// TwinCAT 3 PLC project Untitled1
// ProgramVersion: 3.1.4023.0
// libraries:
//   Tc2_MC2, * (Beckhoff Automation GmbH)
//   Tc2_Standard, * (Beckhoff Automation GmbH)
//   Tc2_System, * (Beckhoff Automation GmbH)
//   Tc3_Module, * (Beckhoff Automation GmbH)
// project tree:
//   DUTs/ st_axisInput.TcDUT, st_axisInterface.TcDUT, st_axisOutput.TcDUT
//   / GlobalTextList.TcGTLO, PlcTask.TcTTO, Visualization Manager.TcVMO (not stored)
//   GVLs/ GVL_Axis.TcGVL
//   POUs/ Fb_Motion.TcPOU, MAIN.TcPOU
//   VISUs/ VISU_1.TcVIS, VISU_2.TcVIS
// real-time tasks:
//   TASK PlcTask: cycle T#10ms, priority 20, ADS port 350
// motion (NC):
//   TASK NC-Task 1 SAF: cycle T#2ms, priority 4, ADS port 501
//   TASK NC-Task 1 SVB: cycle T#10ms, priority 8, ADS port 511
//   AXIS Axis 1 (id 1)
//     OtherSettings: AllowMotionCmdToSlave=true
//     encoder EncType=1
//     drive DrvType=5
//       Analog: TorqueSetpointScale=10, ScaleFactorActTorque=0.1
//     controller CtrType=1
//       CtrPara: PriorControlFactor=1
//         Observer: BandWidth=20
// variable links:
//   Untitled1/Untitled1 Instance <-> NC-Task 1 SAF/Axes/Axis 1
//     PlcTask Inputs/GVL_Axis.Axis1.NcToPlc <-> Outputs/ToPlc
//     PlcTask Outputs/GVL_Axis.Axis1.PlcToNc <-> Inputs/FromPlc

CONFIGURATION Untitled1
    RESOURCE PLC ON TwinCAT3
        TASK PlcTask(INTERVAL := T#10ms, PRIORITY := 20);
        PROGRAM MAIN WITH PlcTask : MAIN;
    END_RESOURCE
END_CONFIGURATION

// ---- DUTs/st_axisInput.TcDUT
TYPE st_axisInput :
STRUCT
	

	bPowerEnable	:	BOOL;
	bMoveAbs		:	BOOL;
	bStop			:	BOOL;
	bReset			:	BOOL;
	
	
	fOverride	:	LREAL;
	fPosition	:	LREAL;
	fVelocity	:	LREAL;

	
	
	

END_STRUCT
END_TYPE

// ---- DUTs/st_axisInterface.TcDUT
TYPE st_axisInterface :
STRUCT
	

IN	:	st_axisInput;
OUT	:	st_axisOutput;


END_STRUCT
END_TYPE

// ---- DUTs/st_axisOutput.TcDUT
TYPE st_axisOutput :
STRUCT
	

	bPowerEnabled	:	BOOL;
	bPowerErr		:	BOOL;

	bMoveAbsDone	:	BOOL;
	bMoveAbsBusy	:	BOOL;
	bMoveAbsErr		:	BOOL;
	
	
	bStopDone		:	BOOL;
	bStopActive		:	BOOL;
	bStopErr		:	BOOL;
	
	bResetDone		:	BOOL;
	bResetErr		:	BOOL;

END_STRUCT
END_TYPE

// ---- GVLs/GVL_Axis.TcGVL
{attribute 'qualified_only'}
VAR_GLOBAL
	

	Axis1	:	AXIS_REF;		//	1. Motor
	
	stAxis1	:	st_axisInterface;
	
	
	Axis2	:	AXIS_REF;		//	2.Motor

	stAxis2	:	st_axisInterface;

END_VAR

// ---- POUs/MAIN.TcPOU
PROGRAM MAIN
VAR
	FbMotion1: Fb_Motion;
	FbMotion2: Fb_Motion;
	nState: INT;
	bButon: BOOL;
	T1: TON;
	T2: TON;
	T3: TON;
	bResetButon	:	BOOL;
	rtrig1: R_TRIG;
	bCounter: BOOL;
	nCounter: INT;
	sMsgInfo: STRING;
	sMsgVelo: STRING;
	sMsgPosition: STRING;
	fPositionVisu: LREAL;
END_VAR



ACT_Motion();
ACT_Visu();







FbMotion1(Axis:=GVL_Axis.Axis1 , stAxis:=GVL_Axis.stAxis1 );
//FbMotion2(Axis:=GVL_Axis.Axis2 , stAxis:=GVL_Axis.stAxis2 );

ACTION ACT_Motion:


rtrig1(CLK:=bCounter , Q=> );


CASE nState OF
	



	0:
	
		IF bButon THEN
			
		GVL_Axis.stAxis1.IN.bPowerEnable	:=	TRUE;
		GVL_Axis.stAxis1.IN.fOverride	:=	100.0;
		GVL_Axis.stAxis1.IN.bStop	:=	FALSE;	
		GVL_Axis.stAxis1.IN.bMoveAbs	:=	FALSE;
		nState := 1;
		
		END_IF
	
		
	1:
		IF	bButon	
		AND NOT GVL_Axis.stAxis1.OUT.bPowerErr
		AND NOT GVL_Axis.stAxis1.OUT.bStopActive 
		AND GVL_Axis.stAxis1.OUT.bPowerEnabled THEN
		
			nState := 10;
			
		END_IF
	
	
	10:
		
		GVL_Axis.stAxis1.IN.fPosition	:=	5000;
		GVL_Axis.stAxis1.IN.fVelocity	:=	650;
		
		GVL_Axis.stAxis1.IN.bMoveAbs	:=	TRUE;
		
		IF GVL_Axis.stAxis1.OUT.bMoveAbsBusy 
		AND NOT GVL_Axis.stAxis1.OUT.bMoveAbsErr	THEN
			
			nState := 20;

		ELSIF 	GVL_Axis.stAxis1.OUT.bMoveAbsErr 
		OR GVL_Axis.stAxis1.OUT.bPowerErr THEN
			
			nState := 999;
		
		END_IF
		
	20:
		sMsgInfo	:=	'Sistem Belirtilen Pozisyona Hareket Etmekte';
		
		IF GVL_Axis.stAxis1.OUT.bMoveAbsDone
		AND NOT GVL_Axis.stAxis1.OUT.bMoveAbsErr THEN
		
			GVL_Axis.stAxis1.IN.bMoveAbs	:=	FALSE;	
			nState := 30;
		
		ELSIF 	GVL_Axis.stAxis1.OUT.bMoveAbsErr 
		OR GVL_Axis.stAxis1.OUT.bPowerErr THEN
			
		nState := 999;
					
		END_IF
		
	
	30:
		
		sMsgInfo	:=	CONCAT(STR1:=TIME_TO_STRING(T1.ET) , STR2:='süredir bekleniyor.' );
	
		T1(IN:= TRUE, PT:=T#5S);
		
		IF T1.Q THEN
			nState := 40;
			T1(IN:= FALSE);
		END_IF
	
	40:
	
	
		GVL_Axis.stAxis1.IN.fPosition	:=	10000;
		GVL_Axis.stAxis1.IN.fVelocity	:=	1000;
		
		GVL_Axis.stAxis1.IN.bMoveAbs	:=	TRUE;
		
		IF GVL_Axis.stAxis1.OUT.bMoveAbsBusy 
		AND NOT GVL_Axis.stAxis1.OUT.bMoveAbsErr	THEN
			
			nState := 50;

		ELSIF 	GVL_Axis.stAxis1.OUT.bMoveAbsErr 
		OR GVL_Axis.stAxis1.OUT.bPowerErr THEN
			
			nState := 999;
		
		END_IF
		
	50:
		sMsgInfo	:=	'Sistem Belirtilen Pozisyona Hareket Etmekte';

		IF GVL_Axis.stAxis1.OUT.bMoveAbsDone
		AND NOT GVL_Axis.stAxis1.OUT.bMoveAbsErr THEN
		
			GVL_Axis.stAxis1.IN.bMoveAbs	:=	FALSE;	
			nState := 60;
		
		ELSIF 	GVL_Axis.stAxis1.OUT.bMoveAbsErr 
		OR GVL_Axis.stAxis1.OUT.bPowerErr THEN
			
		nState := 999;
					
		END_IF
	
	
	60:
		sMsgInfo	:=	'Malzemeler Bekleniyor.';
		IF rtrig1.Q THEN
			nCounter := nCounter + 1;			
		END_IF
		IF nCounter >=6 THEN
			nCounter := 0;
			nState := 70;
		END_IF
		
	70:
		
		GVL_Axis.stAxis1.IN.fPosition	:=	0;
		GVL_Axis.stAxis1.IN.fVelocity	:=	2000;
		
		GVL_Axis.stAxis1.IN.bMoveAbs	:=	TRUE;
		
		IF GVL_Axis.stAxis1.OUT.bMoveAbsBusy 
		AND NOT GVL_Axis.stAxis1.OUT.bMoveAbsErr	THEN
			
			nState := 80;

		ELSIF 	GVL_Axis.stAxis1.OUT.bMoveAbsErr 
		OR GVL_Axis.stAxis1.OUT.bPowerErr THEN
			
			nState := 999;
		
		END_IF
	
	
	80:
		sMsgInfo	:=	'Başlangıç Pozisyonuna Dönülüyor.';
		
		IF GVL_Axis.stAxis1.OUT.bMoveAbsDone
		AND NOT GVL_Axis.stAxis1.OUT.bMoveAbsErr THEN
		
			GVL_Axis.stAxis1.IN.bMoveAbs	:=	FALSE;	
			nState := 90;
		
		ELSIF 	GVL_Axis.stAxis1.OUT.bMoveAbsErr 
		OR GVL_Axis.stAxis1.OUT.bPowerErr THEN
			
		nState := 999;
					
		END_IF
		
	90:
		T3(IN:= TRUE, PT:=T#3S);
		
		IF T3.Q THEN
			nState := 0;
			T3(IN:= FALSE);
		END_IF
	

		
		
	999:
		GVL_Axis.stAxis1.IN.bReset	:=	TRUE;
		
		IF NOT	GVL_Axis.stAxis1.OUT.bResetErr 
		AND GVL_Axis.stAxis1.OUT.bResetDone
		AND bResetButon THEN
	
			nState := 0;
		
		ELSIF	GVL_Axis.stAxis1.OUT.bResetErr THEN
			nState := 1000;
		END_IF
		
		
		
END_CASE



IF NOT bButon THEN
	

	sMsgInfo	:=	'Sistem Kapalı Durumda.';

	T1(IN:= FALSE);
	T2(IN:= FALSE);
	T3(IN:= FALSE);
	
	GVL_Axis.stAxis1.IN.bStop	:=	TRUE;
	
	IF GVL_Axis.stAxis1.OUT.bStopDone
	AND 	GVL_Axis.stAxis1.OUT.bStopActive
	AND NOT	GVL_Axis.stAxis1.OUT.bMoveAbsErr
	AND NOT GVL_Axis.stAxis1.OUT.bPowerErr	 THEN
	
			nState := 0;
		
			GVL_Axis.stAxis1.IN.bPowerEnable	:=	TRUE;
			GVL_Axis.stAxis1.IN.fOverride	:=	100.0;
			
			GVL_Axis.stAxis1.IN.bStop	:=	FALSE;	
	END_IF
	
END_IF
END_ACTION

ACTION ACT_Visu:


sMsgVelo		:=	REAL_TO_STRING(GVL_Axis.Axis1.NcToPlc.ActVelo);
sMsgPosition	:=	REAL_TO_STRING(GVL_Axis.Axis1.NcToPlc.ActPos);


fPositionVisu	:=	GVL_Axis.Axis1.NcToPlc.ActPos/10;
END_ACTION

END_PROGRAM

// ---- POUs/Fb_Motion.TcPOU
FUNCTION_BLOCK Fb_Motion
VAR_INPUT
END_VAR
VAR_OUTPUT
END_VAR
VAR
	mcPower: MC_Power;
	mcMoveAbs: MC_MoveAbsolute;
	mcStop: MC_Stop;
	McReset: MC_Reset;
END_VAR

VAR_IN_OUT
	
	Axis	:	AXIS_REF;
	stAxis	:	st_axisInterface;
	
END_VAR

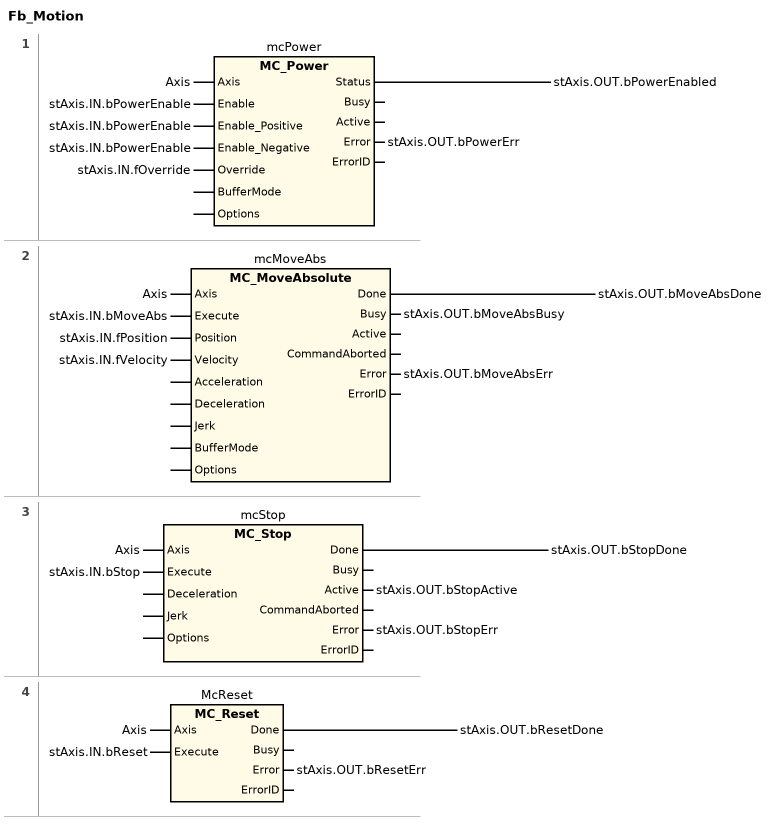
// NETWORK 1
mcPower(
    Axis := Axis,
    Enable := stAxis.IN.bPowerEnable,
    Enable_Positive := stAxis.IN.bPowerEnable,
    Enable_Negative := stAxis.IN.bPowerEnable,
    Override := stAxis.IN.fOverride,
    Error => stAxis.OUT.bPowerErr); // MC_Power
stAxis.OUT.bPowerEnabled := mcPower.Status;

// NETWORK 2
mcMoveAbs(
    Axis := Axis,
    Execute := stAxis.IN.bMoveAbs,
    Position := stAxis.IN.fPosition,
    Velocity := stAxis.IN.fVelocity,
    Busy => stAxis.OUT.bMoveAbsBusy,
    Error => stAxis.OUT.bMoveAbsErr); // MC_MoveAbsolute
stAxis.OUT.bMoveAbsDone := mcMoveAbs.Done;

// NETWORK 3
mcStop(
    Axis := Axis,
    Execute := stAxis.IN.bStop,
    Active => stAxis.OUT.bStopActive,
    Error => stAxis.OUT.bStopErr); // MC_Stop
stAxis.OUT.bStopDone := mcStop.Done;

// NETWORK 4
McReset(Axis := Axis, Execute := stAxis.IN.bReset, Error => stAxis.OUT.bResetErr); // MC_Reset
stAxis.OUT.bResetDone := McReset.Done;

END_FUNCTION_BLOCK

// ---- GlobalTextList.TcGTLO
TEXTLIST GlobalTextList
  766 = '%s'
  470 = '10000'
  33 = '5000'
  595 = 'AbsMoveBusy'
  573 = 'AbsMoveErr'
  345 = 'Anlık Pozisyon Bilgisi:'
  965 = 'AnlıkPozisyon Bilgisi'
  516 = 'AnlıkPozisyon Bilgisi:'
  574 = 'Durum Bilgisi :'
  266 = 'Ekran Değiştir'
  242 = 'Hız Bilgisi:'
  140 = 'Power Enable'
  247 = 'PowerErr'
  370 = 'Sensor Kontrol'
  279 = 'Start/Stop'
  269 = 'Stop'
  255 = 'StopErr'
  603 = 'StopError'
END_TEXTLIST

// ---- VISUs/VISU_1.TcVIS
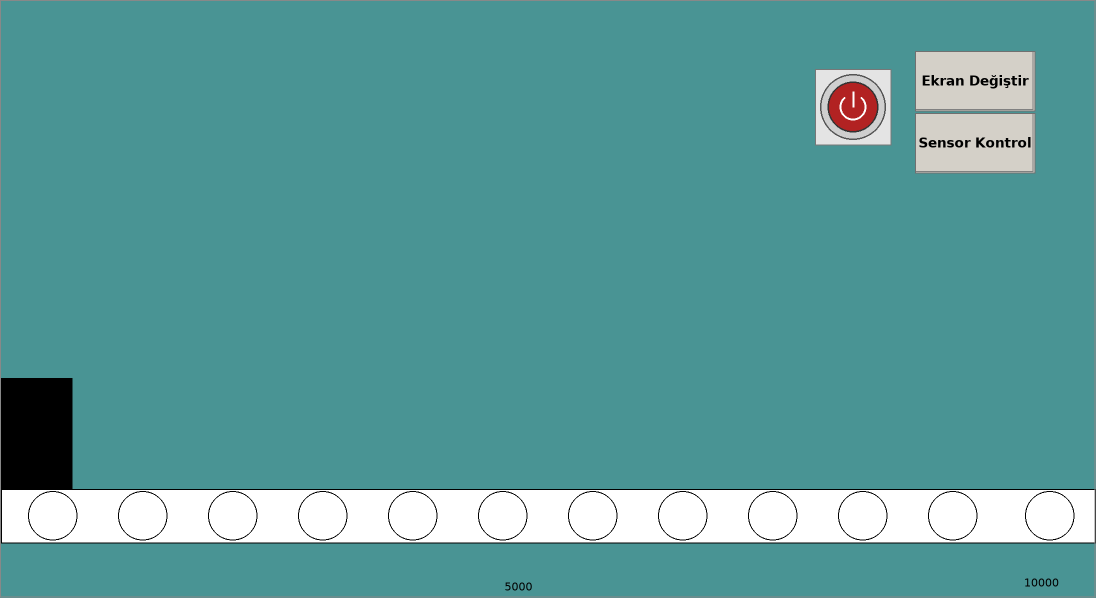
VISUALIZATION VISU_1  // 1096x598
    Rectangle (0,378 72x157)
        p3560616238: MAIN.fPositionVisu
    Group (1,489 1095x54)
        Rectangle (0,0 1095x54)
        Ellipse (27,2 49x49)
        Ellipse (117,2 49x49)
        Ellipse (207,2 49x49)
        Ellipse (297,2 49x49)
        Ellipse (387,2 49x49)
        Ellipse (477,2 49x49)
        Ellipse (567,2 49x49)
        Ellipse (657,2 49x49)
        Ellipse (747,2 49x49)
        Ellipse (837,2 49x49)
        Ellipse (927,2 49x49)
        Ellipse (1024,2 49x49)
    Button (915,51 120x60), "Ekran Değiştir"
        OnMouseClick: change screen: VISU_2
    Button (915,113 120x60), "Sensor Kontrol"
        tap MAIN.bCounter
    PowerSwitch (797,69 112x76), variable: MAIN.bButon, behaviour: TOGGLE, style: Switch-PowerSwitch-Red
    Label (477,576 83x22), "5000"
    Label (1000,572 83x22), "10000"
END_VISUALIZATION

// ---- VISUs/VISU_2.TcVIS
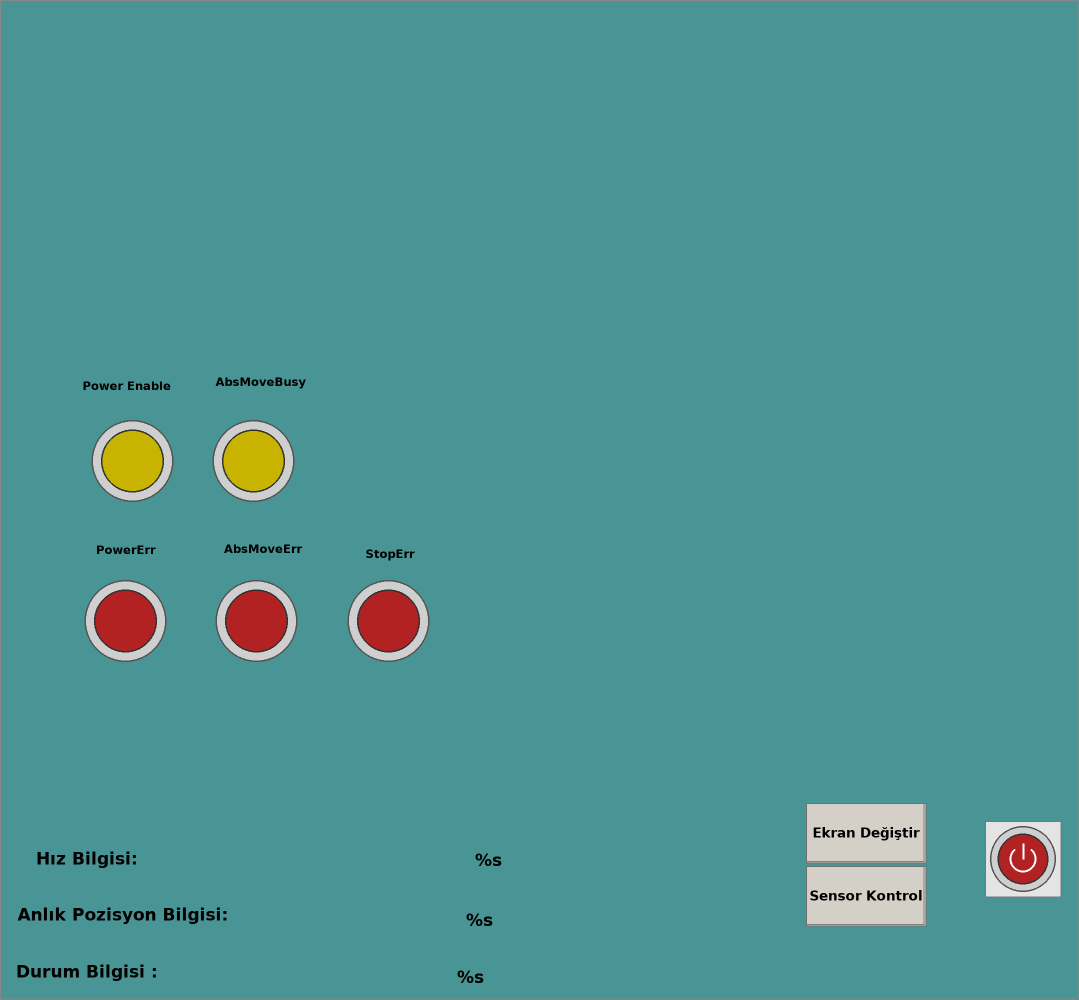
VISUALIZATION VISU_2  // 1079x1000
    Label (3,950 168x43), "Durum Bilgisi :"
    Label (3,893 240x43), "Anlık Pozisyon Bilgisi:"
    Rectangle (240,837 497x46), "%s", text variable: MAIN.sMsgVelo
    Label (3,837 168x43), "Hız Bilgisi:"
    Rectangle (240,897 479x46), "%s", text variable: MAIN.sMsgPosition
    Rectangle (240,954 461x46), "%s", text variable: MAIN.sMsgInfo
    Button (806,803 120x60), "Ekran Değiştir"
        OnMouseClick: change screen: VISU_1
    Button (806,866 120x60), "Sensor Kontrol"
        tap MAIN.bCounter
    PowerSwitch (967,821 112x76), variable: MAIN.bButon, behaviour: TOGGLE, style: Switch-PowerSwitch-Red
    Lamp1 (85,411 95x100), variable: GVL_Axis.stAxis1.OUT.bPowerEnabled, style: Lamp-Lamp1-Yellow
    Lamp1 (206,411 95x100), variable: GVL_Axis.stAxis1.OUT.bMoveAbsBusy, style: Lamp-Lamp1-Yellow
    Lamp1 (78,571 95x100), variable: GVL_Axis.stAxis1.OUT.bPowerErr, style: Lamp-Lamp1-Red
    Lamp1 (209,571 95x100), variable: GVL_Axis.stAxis1.OUT.bMoveAbsErr, style: Lamp-Lamp1-Red
    Lamp1 (341,571 95x100), variable: GVL_Axis.stAxis1.OUT.bStopErr, style: Lamp-Lamp1-Red
    Label (72,372 110x28), "Power Enable"
    Label (206,368 110x28), "AbsMoveBusy"
    Label (335,540 110x28), "StopErr"
    Label (208,535 110x28), "AbsMoveErr"
    Label (71,536 110x28), "PowerErr"
END_VISUALIZATION
